(* PLC project Tc2_Utilities.FB_HashTableCtrl Demo, tc3-libraries-kb TwinCAT 3.1 *)
(* stored: creationDateTime 2026-05-10T20:00:00, modificationDateTime 2026-05-10T20:00:00 *)

PROGRAM P_Demo_FB_HashTableCtrl
  VAR
    fbFB_HashTableCtrl : FB_HashTableCtrl;  (* Tc2_Utilities.FB_HashTableCtrl 实例 *)
    arg_key : DWORD;  (* VAR_INPUT key *)
    arg_putValue : PVOID;  (* VAR_INPUT putValue *)
    arg_putPosPtr : POINTER TO T_HashTableEntry;  (* VAR_INPUT putPosPtr *)
    out_bOk : BOOL;  (* VAR_OUTPUT bOk *)
    out_getValue : PVOID;  (* VAR_OUTPUT getValue *)
    out_getPosPtr : POINTER TO T_HashTableEntry;  (* VAR_OUTPUT getPosPtr *)
    io_hTable : T_HHASHTABLE;  (* VAR_IN_OUT hTable *)
  END_VAR

            // ============================================================
// Tc2_Utilities.FB_HashTableCtrl 演示程序（FB 实例）
// ============================================================
// 验证步骤：
//   1. 引用 Tc2_Utilities（及依赖类型所在库 Tc2_System 等）
//   2. 编译 + 登录
//   3. 按 doc.md 给 arg_* 赋值
//   4. 在线监视 out_* / io_* 输出
// ============================================================

fbFB_HashTableCtrl(
    key := arg_key,
    putValue := arg_putValue,
    putPosPtr := arg_putPosPtr,
    bOk => out_bOk,
    getValue => out_getValue,
    getPosPtr => out_getPosPtr,
    hTable := io_hTable
);

          
END_PROGRAM
